// TIA Portal V20 export
VAR_GLOBAL   // PLC tag table "08_CmInfo"
END_VAR
VAR_GLOBAL CONSTANT   // user constants
   NO_OF_RF_IDENT_DEVICES : USInt := 1;   // SICAR: Anzahl der RF Lesestellen / SICAR: Number of RF readers
   NO_OF_MV_IDENT_DEVICES : USInt := 1;   // SICAR: Anzahl der MV Lesestellen / SICAR: Number of MV readers
   NO_OF_ET200SPMOTORSTARTER : USInt := 1;   // SICAR: Anzahl Motorstarter / SICAR: Number of ET200SP Motorstarter
END_VAR
